{attribute 'qualified_only'}
VAR_GLOBAL
    IN  AT %I* : ARRAY[0..1] OF BOOL;
    OUT AT %I* : ARRAY[0..1] OF BOOL;
END_VAR

(* stored: Version 1.1.0.1
   GVL IO: Id {b97152d1-c0f4-0704-35ec-78de2c66f09d} *)
